FUNCTION_BLOCK GenCyl (* Basic Function Block Type *)
  (* Standard: 61499-2 *)
  (* Version 0.0, 2011-02-26, Majid Sorouri, nxtControl GmbH, Template *)
  (* Compiler header: package fb.rt.pnp; *)
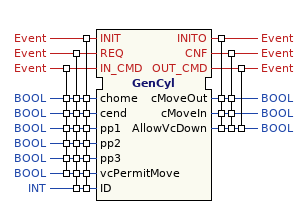
  EVENT_INPUT
    INIT WITH chome, pp1, pp2, pp3, cend, vcPermitMove, ID; (* Initialization Request *)
    REQ WITH chome, cend, pp1, pp2, pp3, vcPermitMove, ID;
    IN_CMD WITH vcPermitMove, pp3, pp2, pp1, cend, chome;
  END_EVENT
  EVENT_OUTPUT
    INITO WITH cMoveOut, cMoveIn, AllowVcDown; (* Initialization Confirm *)
    CNF WITH cMoveOut, cMoveIn, AllowVcDown; (* Execution Confirmation *)
    OUT_CMD WITH AllowVcDown;
  END_EVENT
  VAR_INPUT
    chome : BOOL; (* Input event qualifier *)
    cend : BOOL;
    pp1 : BOOL;
    pp2 : BOOL;
    pp3 : BOOL;
    vcPermitMove : BOOL;
    ID : INT;
  END_VAR
  VAR_OUTPUT
    cMoveOut : BOOL;
    cMoveIn : BOOL;
    AllowVcDown : BOOL;
  END_VAR
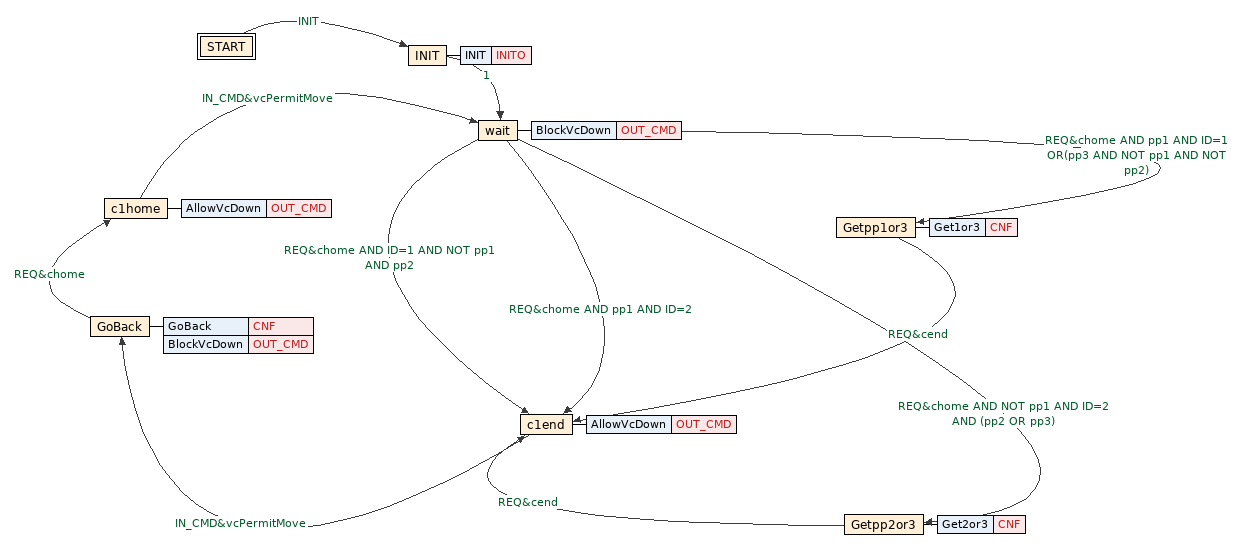
  EC_STATES
    START; (* Initial State *)
    INIT : INIT -> INITO; (* Initialization *)
    c1home : AllowVcDown -> OUT_CMD; (* Normal execution *)
    Getpp1or3 : Get1or3 -> CNF;
    Getpp2or3 : Get2or3 -> CNF;
    GoBack : GoBack -> CNF, BlockVcDown -> OUT_CMD;
    c1end : AllowVcDown -> OUT_CMD;
    wait : BlockVcDown -> OUT_CMD;
  END_STATES
  EC_TRANSITIONS
    START TO INIT := INIT;
    INIT TO wait := 1;
    c1home TO wait := IN_CMD&vcPermitMove;
    c1end TO GoBack := IN_CMD&vcPermitMove;
    GoBack TO c1home := REQ&chome;
    Getpp1or3 TO c1end := REQ&cend;
    wait TO Getpp1or3 := REQ&chome AND pp1 AND ID=1 OR(pp3 AND NOT pp1 AND NOT  pp2);
    wait TO c1end := REQ&chome AND ID=1 AND NOT pp1 AND pp2;
    wait TO Getpp2or3 := REQ&chome AND NOT pp1 AND ID=2 AND (pp2 OR pp3);
    Getpp2or3 TO c1end := REQ&cend;
    wait TO c1end := REQ&chome AND pp1 AND ID=2;
  END_TRANSITIONS
  ALGORITHM INIT IN ST: (* Initialization algorithm *)
cMoveOut:=FALSE;
cMoveIn:=TRUE;
System.out.println("GenCyl INIT " + this);
  END_ALGORITHM
  ALGORITHM REQ IN ST: (* Normally executed algorithm *)
System.out.println("GenCyl REQ " + this);
  END_ALGORITHM
  ALGORITHM Get2or3 IN ST:
cMoveOut:=TRUE;
cMoveIn:=FALSE;
System.out.println("GenCyl Get2or3 " + this);
  END_ALGORITHM
  ALGORITHM Get1or3 IN ST:
cMoveOut:=TRUE;
cMoveIn:=FALSE;
System.out.println("GenCyl Get1or3 " + this);
  END_ALGORITHM
  ALGORITHM GoBack IN ST:
cMoveIn:=TRUE;
cMoveOut:=FALSE;
System.out.println("GenCyl GoBack " + this);
  END_ALGORITHM
  ALGORITHM AllowVcDown IN ST:
AllowVcDown:=TRUE;
System.out.println("GenCyl AllowVcDown " + this);
  END_ALGORITHM
  ALGORITHM BlockVcDown IN ST:
AllowVcDown:=FALSE;
System.out.println("GenCyl BlockVcDown " + this);
  END_ALGORITHM
END_FUNCTION_BLOCK
